FUNCTION_BLOCK FB_ActionList
VAR_INPUT
END_VAR
VAR_OUTPUT
END_VAR
VAR
	pHead	: POINTER TO ST_Pointer;
	pTail	: POINTER TO ST_Pointer;
	pCurrent: POINTER TO ST_Pointer;
	nCount	: UINT;
	pAction : POINTER TO ST_Action;
END_VAR

METHOD M_Add
VAR_INPUT
	stAction : REFERENCE TO ST_Action;
END_VAR

VAR
	pNew : POINTER TO ST_Pointer;
	pAction : POINTER TO ST_Action;
END_VAR
pNew := pHead;
WHILE pNew > 0 DO
	pAction := pNew^.pContent;
	//Action für das Device schon in Liste? Es sei denn, die Action ist bereits schon in Idle versetzt.
	IF (pAction^.eAction >= 50) AND (pAction^.iDevice = stAction.iDevice) AND (pAction^.eAction = stAction.eAction) AND pAction^.eActionStatus <> E_ActionStatus.ACTIONSTATUS_Idle THEN
		RETURN;
	END_IF
	pNew := pNew^.pNext;
END_WHILE

pNew := __NEW(ST_Pointer);
MEMSET(pNew,0,SIZEOF(ST_Pointer));
pAction := __NEW(ST_Action);
MEMCPY(pAction,ADR(stAction),SIZEOF(stAction));
pNew^.pContent := pAction;
IF pHead = 0 THEN
	pHead := pTail := pNew;
ELSE
	pNew^.pPrev := pTail; 
	pTail^.pNext := pNew;
	pTail := pNew;
END_IF
nCount := nCount + 1;
END_METHOD

METHOD M_CleanUp
VAR_INPUT
END_VAR
VAR
	pSeek : POINTER TO ST_Pointer;
	pTemp : POINTER TO ST_Pointer;
	pAction : POINTER TO ST_Action;
END_VAR
//Actions, welche Ready oder in Error gegangen sind in Idle setzen (werden beim nächsten Aufruf gelöscht)
pSeek := pHead;
WHILE (pSeek > 0) DO
	pAction := pSeek^.pContent;
	IF pAction^.eActionStatus = E_ActionStatus.ACTIONSTATUS_Ready OR pAction^.eActionStatus = E_ActionStatus.ACTIONSTATUS_Error THEN
		pAction^.eActionStatus := E_ActionStatus.ACTIONSTATUS_Idle;
		pSeek := pSeek^.pNext;
	ELSIF pAction^.eActionStatus = E_ActionStatus.ACTIONSTATUS_Idle THEN
		IF pSeek = pHead THEN	//Gesuchter ist Head
			IF pSeek^.pNext > 0 THEN //hat Nachfolger
				//Nachfolger wird zum Head
				pHead := pSeek^.pNext;
				pHead^.pPrev := 0; //Head hat keinen Vorgänger
				IF pSeek = pCurrent THEN
					pCurrent := 0;
				END_IF
			ELSE //hat keinen Nachfolger
				pHead := 0;
				pTail := 0;
				pCurrent := 0;				
			END_IF
		ELSIF pSeek = pTail THEN //pSeek ist Tail
			//Vorgänger wird Tail
			pTail := pTail^.pPrev;
			pTail^.pNext := 0; //Tail hat keinen Nachfolger
			IF pSeek = pCurrent THEN
				pCurrent := 0;
			END_IF
		ELSE //pSeek ist in der Mitte
			//Vorgänger beim Nachfolger eintragen
			pTemp := pSeek^.pPrev;
			pTemp^.pNext := pSeek^.pNext;
			//Vorganger beim Nachfolger eintragen
			pTemp := pSeek^.pNext;
			pTemp^.pPrev := pSeek^.pPrev;
			IF pSeek = pCurrent THEN
				pCurrent := pSeek^.pNext;
			END_IF			
		END_IF
		pTemp := pSeek;
		pSeek := pSeek^.pNext;
		__DELETE(pTemp);
		__DELETE(pAction);
		nCount := nCount - 1;		
	ELSE
		pSeek := pSeek^.pNext;
	END_IF
END_WHILE
END_METHOD

METHOD M_GetFromId : POINTER TO ST_Action
VAR_INPUT
	nActionId : UINT;
END_VAR

VAR
	pTemp : POINTER TO ST_Pointer;
	pAction : POINTER TO ST_Action;
END_VAR
pTemp := pHead;
WHILE (pTemp > 0) DO
	pAction := pTemp^.pContent;
	IF pAction^.nActionId = nActionId THEN
		M_GetFromId := pAction;
		RETURN;
	ELSE
		pTemp := pTemp^.pNext;
	END_IF
END_WHILE
END_METHOD

METHOD M_GetNext : POINTER TO ST_Action
VAR_INPUT
END_VAR
IF pCurrent > 0 THEN
	M_GetNext := pCurrent^.pContent;
	pCurrent := pCurrent^.pNext;
END_IF
END_METHOD

METHOD M_Reset
VAR_INPUT
END_VAR

VAR
	pDelete : POINTER TO ST_Pointer;
	pNext	: POINTER TO ST_Pointer;
	pAction : POINTER TO ST_Action;
END_VAR
pDelete := pHead;
WHILE  pDelete > 0 DO
	pAction := pDelete^.pContent;
	pNext := pDelete^.pNext;
	__DELETE(pAction);
	__DELETE(pDelete);
	pDelete := pNext;
END_WHILE
pHead := 0;
pTail := 0;
pCurrent := 0;
nCount := 0;
END_METHOD

METHOD M_SetCurrentToHead
VAR_INPUT
END_VAR
pCurrent := pHead;
END_METHOD

PROPERTY P_bActionsAvailable : BOOL
GET
VAR
	pTemp : POINTER TO ST_Pointer;
	pAction : POINTER TO ST_Action;
END_VAR
//Actions vorhanden die in Active, Pause oder Pause Request sind ?
pTemp := pHead;
WHILE (pTemp > 0) DO
	pAction := pTemp^.pContent;
	IF pAction^.eActionStatus >= E_ActionStatus.ACTIONSTATUS_Active AND pAction^.eActionStatus <= E_ActionStatus.ACTIONSTATUS_Pause THEN
		P_bActionsAvailable := TRUE;
		RETURN;
	ELSE
		pTemp := pTemp^.pNext;
	END_IF
END_WHILE
END_GET
END_PROPERTY

END_FUNCTION_BLOCK

(* stored: Version 1.1.0.1, ProductVersion 3.1.4022.18
   POU FB_ActionList: Id {bacdaf0b-df02-4cab-946f-116c2c59f873}, SpecialFunc None
   Method M_Add: Id {687a756e-ae44-478f-bd6d-40372b486ff4}
   Method M_CleanUp: Id {46a07fb6-d3be-4bbe-84dd-5ef3b3784531}
   Method M_GetFromId: Id {43f37ace-69c8-42bb-90f5-e2b9c18d08eb}
   Method M_GetNext: Id {9d6fb1e0-1263-4fca-94c5-4bb3875e2559}
   Method M_Reset: Id {27377d0f-816d-4bd3-99ad-496f9d533ca2}
   Method M_SetCurrentToHead: Id {42f4134a-553c-434c-945c-2dc22e7172fe}
   Property P_bActionsAvailable: Id {792cdb94-b6e8-4a4f-959f-c5da98f11706}
   Get Get: Id {e281ba32-670d-437b-9753-34fe9cd1165c} *)
